  MoveL 3715 to (49.53, -23.85, 160) mm, rotated rx 180 ry 0 rz 180 deg; joints [-165.618, -46.193, -89.495, 19.715, 47.415, -13.631]
  Call Extruder(137.23498)
  MoveL 3716 to (53.59, -12.23, 160) mm, rotated rx -180 ry 0 rz -180 deg; joints [-164.2, -46.785, -88.193, 21.818, 47.105, -15.243]
  Call Extruder(148.16520)
  MoveL 3717 to (54.97, 0, 160) mm, rotated rx -180 ry 0 rz 180 deg; joints [-162.641, -47.2, -87.284, 24.043, 47.082, -16.898]
  Call Extruder(159.09542)
  MoveL 3718 to (53.59, 12.23, 160) mm, rotated rx -180 ry 0 rz 180 deg; joints [-160.996, -47.418, -86.807, 26.279, 47.348, -18.498]
  Call Extruder(170.02557)
  MoveL 3719 to (49.52, 23.85, 160) mm, rotated rx 180 ry 0 rz -180 deg; joints [-159.322, -47.428, -86.785, 28.424, 47.888, -19.948]
  Call Extruder(180.95584)
  MoveL 3720 to (42.98, 34.27, 160) mm, rotated rx 180 ry 0 rz 180 deg; joints [-157.673, -47.231, -87.217, 30.391, 48.672, -21.171]
  Call Extruder(191.88597)
  MoveL 3721 to (34.27, 42.98, 160) mm, rotated rx -180 ry 0 rz -180 deg; joints [-156.102, -46.834, -88.084, 32.109, 49.654, -22.11]
  Call Extruder(202.81624)
  MoveL 3722 to (23.85, 49.53, 160) mm, rotated rx 180 ry 0 rz -180 deg; joints [-154.667, -46.259, -89.349, 33.524, 50.781, -22.728]
  Call Extruder(213.74639)
  MoveL 3723 to (12.23, 53.59, 160) mm, rotated rx 180 ry 0 rz 180 deg; joints [-153.426, -45.532, -90.958, 34.594, 51.993, -23.01]
  Call Extruder(224.67661)
  MoveL 3724 to (0, 54.97, 160) mm, rotated rx -180 ry 0 rz 180 deg; joints [-152.438, -44.688, -92.838, 35.285, 53.229, -22.958]
  Call Extruder(235.60683)
  MoveL 3725 to (-12.23, 53.59, 160) mm, rotated rx 180 ry 0 rz 180 deg; joints [-151.764, -43.769, -94.908, 35.567, 54.427, -22.586]
  Call Extruder(246.53697)
  MoveL 3726 to (-23.85, 49.52, 160) mm, rotated rx 180 ry 0 rz 180 deg; joints [-151.463, -42.818, -97.072, 35.413, 55.529, -21.921]
  Call Extruder(257.46725)
  MoveL 3727 to (-34.27, 42.98, 160) mm, rotated rx 180 ry 0 rz 180 deg; joints [-151.589, -41.884, -99.228, 34.798, 56.483, -20.994]
  Call Extruder(268.39737)
  MoveL 3728 to (-42.98, 34.27, 160) mm, rotated rx 180 ry 0 rz -180 deg; joints [-152.179, -41.012, -101.268, 33.708, 57.242, -19.848]
  Call Extruder(279.32765)
  MoveL 3729 to (-49.52, 23.85, 160) mm, rotated rx 180 ry 0 rz 180 deg; joints [-153.248, -40.247, -103.082, 32.149, 57.772, -18.529]
  Call Extruder(290.25779)
  MoveL 3730 to (-53.59, 12.23, 160) mm, rotated rx 180 ry 0 rz 180 deg; joints [-154.769, -39.631, -104.563, 30.158, 58.047, -17.092]
  Call Extruder(301.18801)
  MoveL 3731 to (-54.97, 0, 160) mm, rotated rx 180 ry 0 rz -180 deg; joints [-156.673, -39.197, -105.62, 27.817, 58.056, -15.598]
  Call Extruder(306.71363)
  MoveL 3732 to (-54.27, -6.18, 160) mm, rotated rx 180 ry 0 rz 180 deg; joints [-157.76, -39.077, -105.913, 26.53, 57.924, -14.849]
  Set speed (130.0 mm/s)
  MoveL 3733 to (-49.9, -9.51, 160) mm, rotated rx 180 ry 0 rz 180 deg; joints [-158.616, -39.27, -105.44, 25.628, 57.457, -14.47]
  Call Extruder(304.71363)
  Set speed (40.0 mm/s)
  MoveL 3734 to (-49.9, -9.51, 160) mm, rotated rx 180 ry 0 rz 180 deg; joints [-158.616, -39.27, -105.44, 25.628, 57.457, -14.47]
  Call Extruder(0.00000)
  Set speed (130.0 mm/s)
  MoveL 3735 to (-4.91, 13.82, 160) mm, rotated rx 180 ry 0 rz 180 deg; joints [-157.786, -42.958, -96.752, 28.163, 53.226, -17.771]
  Call Extruder(2.00000)
  Set speed (40.0 mm/s)
  MoveL 3736 to (-4.91, 13.82, 160) mm, rotated rx 180 ry 0 rz 180 deg; joints [-157.786, -42.958, -96.752, 28.163, 53.226, -17.771]
  Call Extruder(35.17502)
  Set speed (15.0 mm/s)
  MoveL 3737 to (-13.82, 4.92, 160) mm, rotated rx 180 ry 0 rz 180 deg; joints [-158.572, -42.073, -98.789, 26.839, 54.016, -16.557]
  Call Extruder(104.98163)
  MoveL 3738 to (4.92, -13.82, 160) mm, rotated rx 180 ry 0 rz 180 deg; joints [-162.368, -42.945, -96.783, 22.615, 51.972, -14.393]
  Call Extruder(138.15665)
  MoveL 3739 to (13.82, -4.91, 160) mm, rotated rx 180 ry 0 rz 180 deg; joints [-161.491, -43.825, -94.782, 24.049, 51.169, -15.633]
  Call Extruder(136.15665)
  Set speed (40.0 mm/s)
  MoveL 3740 to (13.82, -4.91, 160) mm, rotated rx 180 ry 0 rz 180 deg; joints [-161.491, -43.825, -94.782, 24.049, 51.169, -15.633]
  Set speed (1000.0 mm/s)
  Call Extruder(-1)
  MoveL 3741 to (13.82, -4.91, 160) mm, rotated rx 180 ry 0 rz 180 deg; joints [-161.491, -43.825, -94.782, 24.049, 51.169, -15.633]
  Call Extruder(0.00000)

--- Python program Extruder ---
# This macro allows simulating a 3D printing extruder
# The macro will output spray gun statistics
#
# More information about the RoboDK API here:
# https://robodk.com/doc/en/RoboDK-API.html
# For more information visit:
# http://www.robodk.com/doc/en/PythonAPI/robolink.html
#
# Define the default action (0 to deactivate, +1 to activate, -1 to clear any spray gun simulation)
# Setting it to None will display a message
ACTION = None
# Check if we are running this program inside another program and passing arguments
import sys
if len(sys.argv) > 1:
    ACTION = float(sys.argv[1])
    # For faster speed: igone values greater than 0
    if ACTION > 0:
        quit()

from robolink import *    # API to communicate with RoboDK
from robodk import *      # basic matrix operations
RDK = Robolink()

# quit if we are not in simulation mode
if RDK.RunMode() != RUNMODE_SIMULATE:
    quit()

# Get any previously added spray gun simulations and display statistics (spray on the part vs spray falling out of the part)
existing_material_simulation = False
info, stats_data = RDK.Spray_GetStats()
if stats_data.size(1) > 0:
    print("Spray gun statistics:")
    print(info)
    print(stats_data.tr())
    existing_material_simulation = True
    # # Diplay statistics
    # RDK.ShowMessage("Material used: %.1f%%<br>Material waisted: %.1f%%<br>Total particles: %.1f" % (data[1,0],data[2,0],data[3,0]), True)
    # # Clear previous spray
    # RDK.Spray_Clear()

# If the default ACTION is None, display a message to activate/deactivate the spray gun
if ACTION is None:
    print('Note: This macro can be called as Extruder(0) to turn it ON or Extruder(-1) to turn it OFF')
    entry = mbox('Turn Extruder ON or OFF', ('On', '0'), ('Off', '-1'))
    if not entry:
        quit()
    ACTION = int(entry)

if ACTION < 0:
    # Turn material deposition off
    # Select Escape to delete existing material simulations
    #RDK.Spray_Clear()
    RDK.Spray_SetState(SPRAY_OFF)

elif ACTION >= 0:

    if existing_material_simulation:
        # Select Esc key to delete existing material simulations and force a new type of spray gun simulation
        RDK.Spray_SetState(SPRAY_ON)
        exit()


    # Create a new spray gun object in RoboDK for material deposition (3D printing simulation)
    # by using RDK.Spray_Add(tool, object, options_command, volume, geometry)
    # tool: tool item (TCP) to use
    # object: object to project the particles
    # options_command (optional): string to specify options. Example:
    #     STEP=AxB: Defines the grid to be projected 1x1 means only one line of particle projection (for example, for welding)
    #     PARTICLE: Defines the shape and size of particle (sphere or particle), unless a specific geometry is provided:
    #       a- SPHERE(radius, facets)
    #       b- SPHERE(radius, facets, scalex, scaley, scalez)
    #       b- CUBE(sizex, sizey, sizez)
    #     RAND=factor: Defines a random factor factor 0 means that the particles are not deposited randomly
    #     ELLYPSE: defines the volume as an ellypse (default)
    #     RECTANGLE: defines the volume as a rectangle
    #     PROJECT: project the particles to the surface (default) (for welding, painting or scanning)
    #     NO_PROJECT: does not project the particles to the surface (for example, for 3D printing)
    #
    # volume (optional): Matrix of parameters defining the volume of the spray gun
    # geometry (optional): Matrix of vertices defining the triangles.


    diameter = 22.225 # in mm
    detail = 8 # number of rings of detail to display the sphere
    scale = '1,1,0.5' # scale the particle in 0.5 along the tool Z axis (simulating gravity effect)
    options_command = "ELLYPSE NO_PROJECT PARTICLE=SPHERE(%.3f,%.0f,%s)" % (diameter, detail, scale) # simulate
    #options_command = "PARTICLE=CUBE(10,10,2) STEP=8x8"
    #options_command = "PARTICLE=SPHERE(4,8) STEP=8x8"
    #options_command = "PARTICLE=SPHERE(4,8,1,1,0.1) STEP=8x8 RAND=3"

    # Example commands for welding:
    # options_command = "PROJECT PARTICLE=SPHERE(4,8)"
    # options_command = PARTICLE=SPHERE(4,8) STEP=1x0

    tool = 0    # auto detect active tool
    obj = 0     # auto detect object in active reference frame

    # Material is deposited at 0,0,0 with respect to the TCP coordinates
    close_param = [0,0,0,  0,0,0,  0,0,0,     0.7,0.5,0.8,1] # color as RGBA
    far_param   = [0,0,0,  0,0,0,  0,0,0,     0.7,0.5,0.8,1] # color as RGBA
    volume = Mat([close_param, far_param])
    RDK.Spray_Add(tool, obj, options_command, volume.tr())
    RDK.Spray_SetState(SPRAY_ON)

--- Python program SimulateFinalResult ---
# This script will simulate the final result of the 3D printed part using the Spray function

# Or visit: http://www.robodk.com/doc/PythonAPI/
# Note: you do not need to keep a copy of this file, your python script is saved with the station
from robolink import *    # API to communicate with RoboDK
from robodk import *      # basic matrix operations


RENDER = True      # Set to False
STEP_MM = 2         # Detail step in MM for linear moves
STEP_DEG = 2        # Detail step in DEG for joint moves

# Start a connection with the RoboDK API
RDK = Robolink()

# Select the first/only robot in the cell:
program = RDK.ItemUserPick('Select a program to simulate', ITEM_TYPE_PROGRAM)
if not program.Valid():
    raise Exception("No program available")

# Get the robot
robot = RDK.Item('', ITEM_TYPE_ROBOT)
#robot = program.getLink(ITEM_TYPE_ROBOT) # available in newer versions
if not robot.Valid():
    raise Exception("No robot available")

progname = program.Name()
print("Using program %s" % progname)


# Get the program as a list of joint values
tool = robot.getLink(ITEM_TYPE_TOOL)
progok_jlist = program.InstructionListJoints(STEP_MM, STEP_DEG)
progok = progok_jlist[0] # progok: String that indicates if there are any issues with the program
jlist = progok_jlist[1]  # jlist: list of joints

# Check that the program is correct and has at least a movement
njoints = jlist.size(1)
if njoints < 1:
    raise Exception("Program %s has no movements" % name)

# Check if there are any issues with the program:
if progok != "Success":
    raise Exception("Problems with program %s: %s." %(name, progok))

# Reset any material deposition simulation
RDK.Spray_Clear()

robot.setPoseTool(tool)

# Start material deposition simulation according to the Extruder script
RDK.RunProgram('Extruder(0)')
# Alternatively:
#RDK.Item('Extruder', ITEM_TYPE_PYTHON).RunProgram([1])

if not RENDER:
    RDK.Render(False)

# Iterate through all joints in the matrix and check for collisions
njoints_all = jlist.size(1)
for i in range(njoints_all):
    ji = jlist[:,i].tolist()

    # Update the robot to a new position (it will create a new particle)
    robot.setJoints(ji)
    if not RENDER:
        # If Render is turned off (faster) update the position to draw a new particle
        RDK.Update()

    # Show a message in the RoboDK status bar from time to time
    if i % 10 == 0:
        msg = "Quick material deposition simulation for %s (%.1f %%)" % (progname, 100.0*(i/njoints_all))
        print(msg)
        RDK.ShowMessage(msg, False)

    # Render from time to time even if we have render deactivated
    if not RENDER and i % 500 == 0:
        RDK.Render()

RDK.Render(True)
msg = "Done"
print("Done")
RDK.ShowMessage(msg, False)
